// TIA Portal V17 export
// export: Created 2024-09-02T12:50:16.6708388Z, ExportSetting WithDefaults, DisplayName Totally Integrated Automation Portal, DisplayVersion V17, DisplayName TIA Portal Openness, DisplayVersion V17, DisplayName TIA Portal Version Control Interface, DisplayVersion V17, DisplayName STEP 7 Professional, DisplayVersion V17, DisplayName STEP 7 Safety, DisplayVersion V17, DisplayName WinCC Professional, DisplayVersion V17
DATA_BLOCK "AnwDB_EKS_Data_OP70"   // DB63
{ S7_Optimized_Access := 'TRUE'; DB_Accessible_From_OPC_UA := 'FALSE' }
AUTHOR : VAF
FAMILY : SK
NAME : SK
VERSION : 0.1
// stored: AutoNumber false, DBAccessibleFromOPCUA false, IsOnlyStoredInLoadMemory false, IsRetainMemResEnabled false, IsWriteProtectedInAS false, MemoryReserve 0
   VAR
      EKS1 { ExternalWritable := 'False'} : Struct
         LEVEL { ExternalWritable := 'False'} : Int := 0;   // Schutzstufe / Protection
         LEVEL_1_BE { ExternalWritable := 'False'} : Bool;   // Schutzstufe 1 - Rot Administrator (Level 1) / Protection Level 1 - BLue Maintenance engineering + machine supplier(Level 1)
         LEVEL_3_RD { ExternalWritable := 'False'} : Bool;   // Schutzstufe 1 - Rot Administrator (Level 1) / Protection Level 3 - Red Maintenance technicians (Level 3)
         LEVEL_4_GN { ExternalWritable := 'False'} : Bool := false;   // Schutzstufe 4 - Grün Einrichter (Level 4) / Protection Level 4 - Green Advanced Operator (Level 4)
         LEVEL_5_BK { ExternalWritable := 'False'} : Bool;   // Schutzstufe 6 - Schwarz Bediener (Level 6) / Protection Level 5 - Black Operator (Level 5)
         LIVEDATE { ExternalWritable := 'False'; S7_SetPoint := 'True'} : "TypeKeyData";   // KEY aktuelle Daten / KEY current data
         SAVEDATE { ExternalWritable := 'False'; S7_SetPoint := 'True'} : "TypeKeyData";   // KEY letzte Daten / KEY last data
      END_STRUCT;
   END_VAR
BEGIN
END_DATA_BLOCK
